// TIA Portal V20 export
// export: Created 2025-12-01T14:56:58.3126404Z, ExportSetting None, DisplayName Totally Integrated Automation Portal, DisplayVersion V20 Update 3, DisplayName TIA Portal Openness, DisplayVersion V20 Update 3, DisplayName TIA Portal Version Control Interface, DisplayVersion V20 Update 3, DisplayName STEP 7 Professional, DisplayVersion V20 Update 3, DisplayName STEP 7 Safety, DisplayVersion V20 Update 2, DisplayName WinCC Basic/Comfort/Advanced, DisplayVersion V20 Update 3, DisplayName WinCC Professional, DisplayVersion V20 Update 3, DisplayName WinCC Unified, DisplayVersion V20 Update 3
FUNCTION_BLOCK "FB87_GALIBO_3Frontales"   // FB87, LAD
TITLE = Galibo de 3 Desplomes Frontales (2024)
{ S7_Optimized_Access := 'FALSE' }
AUTHOR : GALIBO
NAME : 20140101
VERSION : 3.0
// stored: AutoNumber false, SetENOAutomatically false
   VAR_INPUT
      Mesa : UInt;
      NumGalibo : UInt;
      EnRodillos : Bool;
      pHs_LecturaDelantera_Des1 : Bool;
      pHs_LecturaTrasera_Des1 : Bool;
      pHs_LecturaDelantera_Des2 : Bool;
      pHs_LecturaTrasera_Des2 : Bool;
      pHs_LecturaDelantera_Error : Bool;
      pHs_LecturaTrasera_Error : Bool;
      pHs_Frontal_1 : Bool;
      pHs_Frontal_2 : Bool;
      pHs_Frontal_3 : Bool;
      HabilitarLectura : Bool;
      PermisoLectura : Bool;
      Rearmar_ConMesaLibre : Bool;
      Numero_Desplomes_2 : Bool;
      Numero_Desplomes_3 : Bool;
   END_VAR
   VAR_OUTPUT
      Baliza : Bool;
      ErrorFrontal : Bool;
      FinLectura : Bool;
   END_VAR
   VAR
      GAL_ET00 : Bool;
      GAL_ET01 : Bool;
      GAL_ET02 : Bool;
      GAL_ET03 : Bool;
      GAL_ET04 : Bool;
      pHsGalibo_OK { ExternalAccessible := 'False'; ExternalVisible := 'False'; ExternalWritable := 'False'} : Bool;
      pHsFrontal_OK : Bool;
      CaraDelantera_Des_PEQUEÑO_NOK : Bool;
      CaraTrasera_Des_PEQUEÑO_NOK : Bool;
      CaraDelantera_Des_MEDIANO_NOK : Bool;
      CaraTrasera_Des_MEDIANO_NOK : Bool;
      CaraDelantera_Des_NOK : Bool;
      CaraTrasera_Des_NOK : Bool;
      CodigoLargura : SInt;
      MemoCodigo : Word;
      STAT_Baliza_Galibo : Bool;
   END_VAR
   VAR_TEMP
      EstadoZona : "EstadoZona";
      EstadoVI : "EstadosMesa";
   END_VAR
   VAR_TEMP   // added for the SCL form of the ladder/FBD networks
      _w1 : Bool;
   END_VAR
BEGIN

REGION Network 1: INICIALIZAR - Recoger las Variables de Estado de la Mesa
   // Se recoge - Estado_CBx
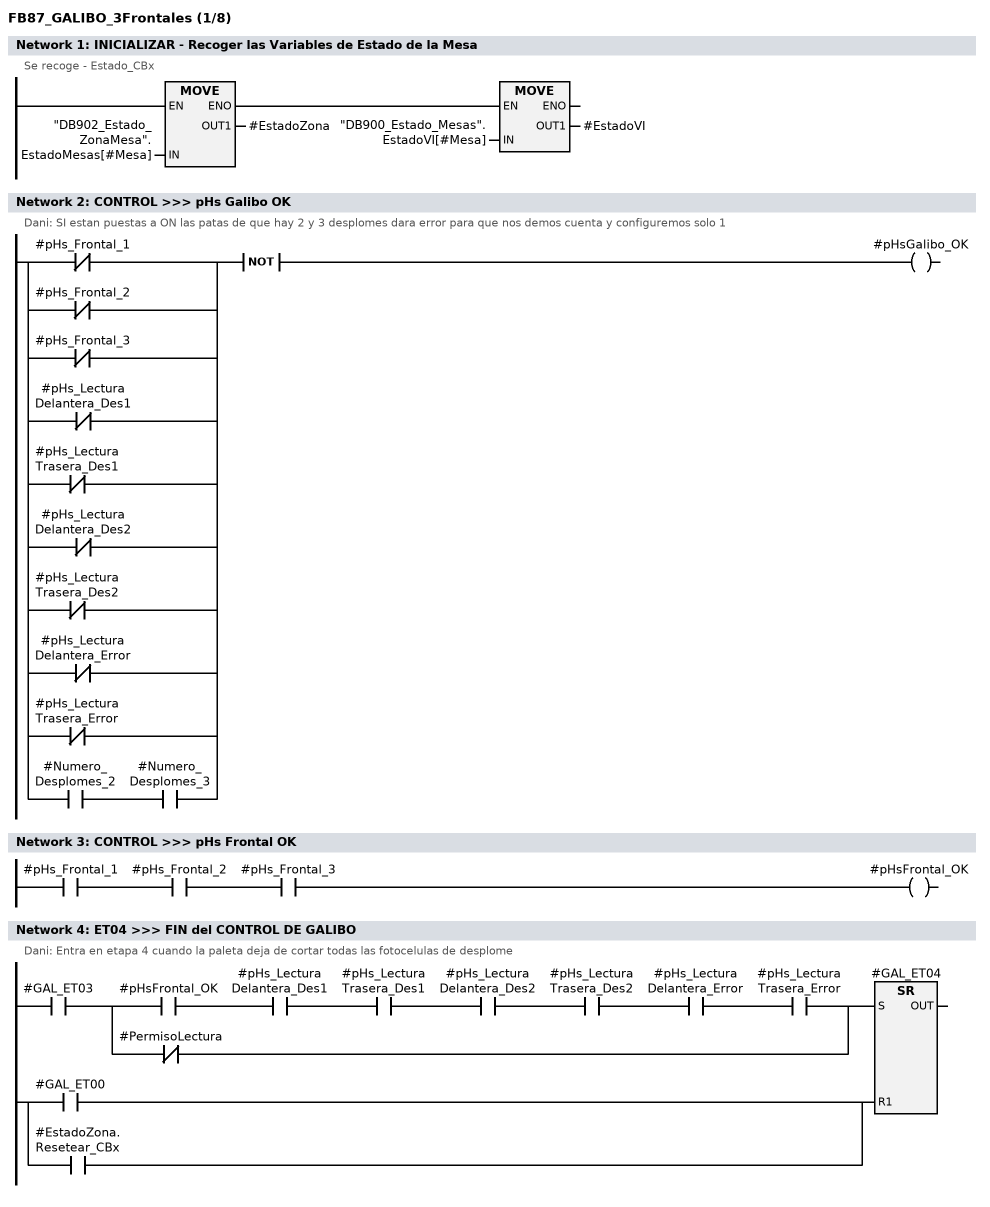
   RUNG wire#powerrail
      Move(in := "DB902_Estado_ZonaMesa".EstadoMesas[#Mesa], out1 => #EstadoZona)
      Move(in := "DB900_Estado_Mesas".EstadoVI[#Mesa], out1 => #EstadoVI)
   END_RUNG
   // the same network as SCL:
   #EstadoZona := "DB902_Estado_ZonaMesa".EstadoMesas[#Mesa];
   #EstadoVI := "DB900_Estado_Mesas".EstadoVI[#Mesa];
END_REGION

REGION Network 2: CONTROL >>> pHs Galibo OK
   // Dani: SI estan puestas a ON las patas de que hay 2 y 3 desplomes dara error para que nos demos cuenta y configuremos solo 1
   RUNG wire#powerrail
      I_Contact( #pHs_Frontal_1 )
      wire#w1
      Not()
      Coil( #pHsGalibo_OK )
   END_RUNG
   RUNG wire#powerrail
      I_Contact( #pHs_Frontal_2 )
   END_RUNG wire#w1
   RUNG wire#powerrail
      I_Contact( #pHs_Frontal_3 )
   END_RUNG wire#w1
   RUNG wire#powerrail
      I_Contact( #pHs_LecturaDelantera_Des1 )
   END_RUNG wire#w1
   RUNG wire#powerrail
      I_Contact( #pHs_LecturaTrasera_Des1 )
   END_RUNG wire#w1
   RUNG wire#powerrail
      I_Contact( #pHs_LecturaDelantera_Des2 )
   END_RUNG wire#w1
   RUNG wire#powerrail
      I_Contact( #pHs_LecturaTrasera_Des2 )
   END_RUNG wire#w1
   RUNG wire#powerrail
      I_Contact( #pHs_LecturaDelantera_Error )
   END_RUNG wire#w1
   RUNG wire#powerrail
      I_Contact( #pHs_LecturaTrasera_Error )
   END_RUNG wire#w1
   RUNG wire#powerrail
      Contact( #Numero_Desplomes_2 )
      Contact( #Numero_Desplomes_3 )
   END_RUNG wire#w1
   // the same network as SCL:
   #pHsGalibo_OK := NOT (NOT #pHs_Frontal_1 OR NOT #pHs_Frontal_2 OR NOT #pHs_Frontal_3 OR NOT #pHs_LecturaDelantera_Des1 OR NOT #pHs_LecturaTrasera_Des1 OR NOT #pHs_LecturaDelantera_Des2 OR NOT #pHs_LecturaTrasera_Des2 OR NOT #pHs_LecturaDelantera_Error OR NOT #pHs_LecturaTrasera_Error OR (#Numero_Desplomes_2 AND #Numero_Desplomes_3));
END_REGION

REGION Network 3: CONTROL >>> pHs Frontal OK
   RUNG wire#powerrail
      Contact( #pHs_Frontal_1 )
      Contact( #pHs_Frontal_2 )
      Contact( #pHs_Frontal_3 )
      Coil( #pHsFrontal_OK )
   END_RUNG
   // the same network as SCL:
   #pHsFrontal_OK := #pHs_Frontal_1 AND #pHs_Frontal_2 AND #pHs_Frontal_3;
END_REGION

REGION Network 4: ET04 >>> FIN del CONTROL DE GALIBO
   // Dani: Entra en etapa 4 cuando la paleta deja de cortar todas las fotocelulas de desplome
   RUNG wire#powerrail
      Contact( #GAL_ET03 )
      wire#w1
      Contact( #pHsFrontal_OK )
      Contact( #pHs_LecturaDelantera_Des1 )
      Contact( #pHs_LecturaTrasera_Des1 )
      Contact( #pHs_LecturaDelantera_Des2 )
      Contact( #pHs_LecturaTrasera_Des2 )
      Contact( #pHs_LecturaDelantera_Error )
      Contact( #pHs_LecturaTrasera_Error )
      wire#w2
      S_SR(operand := #GAL_ET04, r1 := wire#w3)
   END_RUNG
   RUNG wire#w1
      I_Contact( #PermisoLectura )
   END_RUNG wire#w2
   RUNG wire#powerrail
      Contact( #GAL_ET00 )
   END_RUNG wire#w3
   RUNG wire#powerrail
      Contact( #EstadoZona.Resetear_CBx )
   END_RUNG wire#w3
   // the same network as SCL:
   IF #GAL_ET03 AND ((#pHsFrontal_OK AND #pHs_LecturaDelantera_Des1 AND #pHs_LecturaTrasera_Des1 AND #pHs_LecturaDelantera_Des2 AND #pHs_LecturaTrasera_Des2 AND #pHs_LecturaDelantera_Error AND #pHs_LecturaTrasera_Error) OR NOT #PermisoLectura) THEN
       #GAL_ET04 := TRUE;   // SR flip-flop
   END_IF;
   IF #GAL_ET00 OR #EstadoZona.Resetear_CBx THEN #GAL_ET04 := FALSE; END_IF;
END_REGION

REGION Network 5: ET03 >>> Lectura de CARA TRASERA
   // Dani: Entra en etapa 3 cuando la paleta corta una de las fotocelula de desplomeque esten configuradas
   // En la fotocelula error siempre estara metido el desplome mayor tengamos 1, 2 o 3 desplomes
   // En la fotocelula desplome 2 solo tendremos metido el desplome mediano si el numero de desplome es 3
   // En la fotocelula desplome 1 tendremos metido el desplome mas pequeño si el numero de desplome es 2 o 3.
   // Como los desplomes que no existan estaran siempre a ON no hace falta programar ningun tipo de logica para saber cuando se corta la primera
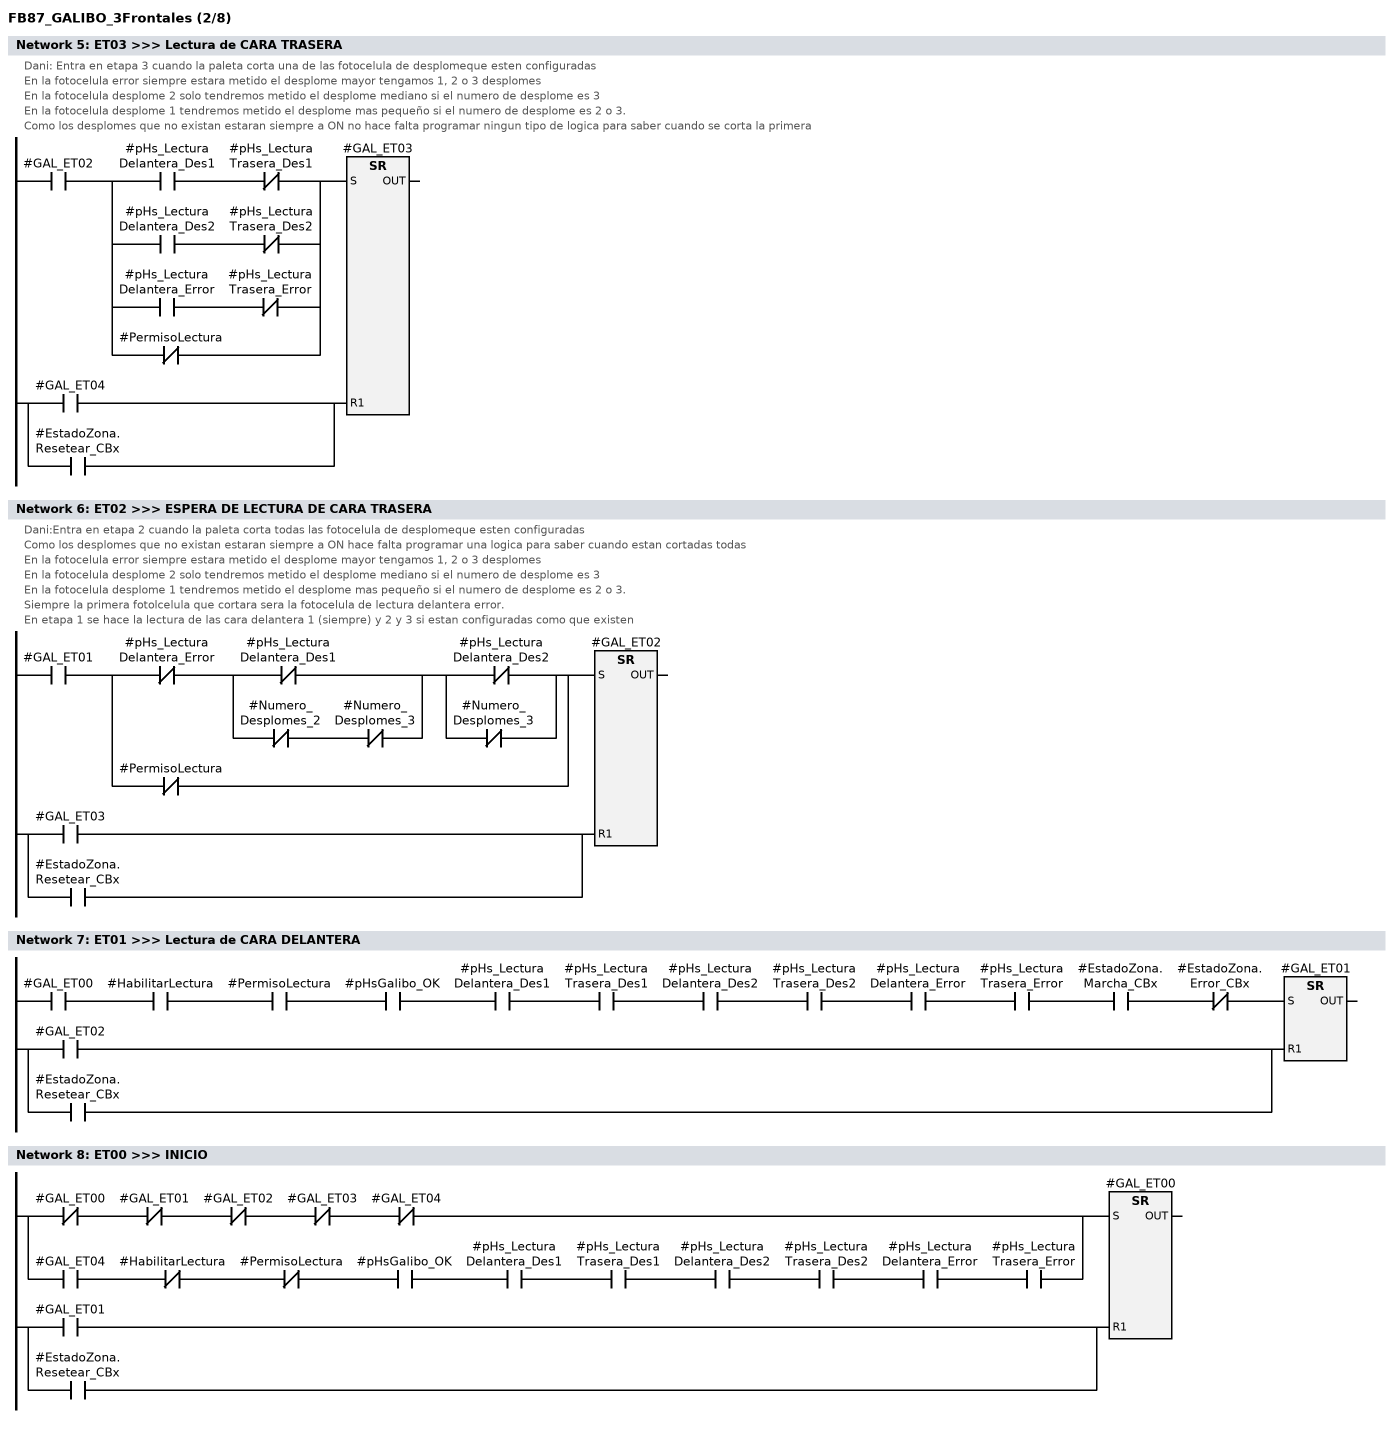
   RUNG wire#powerrail
      Contact( #GAL_ET02 )
      wire#w1
      Contact( #pHs_LecturaDelantera_Des1 )
      I_Contact( #pHs_LecturaTrasera_Des1 )
      wire#w2
      S_SR(operand := #GAL_ET03, r1 := wire#w3)
   END_RUNG
   RUNG wire#w1
      Contact( #pHs_LecturaDelantera_Des2 )
      I_Contact( #pHs_LecturaTrasera_Des2 )
   END_RUNG wire#w2
   RUNG wire#w1
      Contact( #pHs_LecturaDelantera_Error )
      I_Contact( #pHs_LecturaTrasera_Error )
   END_RUNG wire#w2
   RUNG wire#w1
      I_Contact( #PermisoLectura )
   END_RUNG wire#w2
   RUNG wire#powerrail
      Contact( #GAL_ET04 )
   END_RUNG wire#w3
   RUNG wire#powerrail
      Contact( #EstadoZona.Resetear_CBx )
   END_RUNG wire#w3
   // the same network as SCL:
   IF #GAL_ET02 AND ((#pHs_LecturaDelantera_Des1 AND NOT #pHs_LecturaTrasera_Des1) OR (#pHs_LecturaDelantera_Des2 AND NOT #pHs_LecturaTrasera_Des2) OR (#pHs_LecturaDelantera_Error AND NOT #pHs_LecturaTrasera_Error) OR NOT #PermisoLectura) THEN
       #GAL_ET03 := TRUE;   // SR flip-flop
   END_IF;
   IF #GAL_ET04 OR #EstadoZona.Resetear_CBx THEN #GAL_ET03 := FALSE; END_IF;
END_REGION

REGION Network 6: ET02 >>> ESPERA DE LECTURA DE CARA TRASERA
   // Dani:Entra en etapa 2 cuando la paleta corta todas las fotocelula de desplomeque esten configuradas
   // Como los desplomes que no existan estaran siempre a ON hace falta programar una logica para saber cuando estan cortadas todas
   // En la fotocelula error siempre estara metido el desplome mayor tengamos 1, 2 o 3 desplomes
   // En la fotocelula desplome 2 solo tendremos metido el desplome mediano si el numero de desplome es 3
   // En la fotocelula desplome 1 tendremos metido el desplome mas pequeño si el numero de desplome es 2 o 3.
   // Siempre la primera fotolcelula que cortara sera la fotocelula de lectura delantera error.
   // En etapa 1 se hace la lectura de las cara delantera 1 (siempre) y 2 y 3 si estan configuradas como que existen
   RUNG wire#powerrail
      Contact( #GAL_ET01 )
      wire#w1
      I_Contact( #pHs_LecturaDelantera_Error )
      wire#w2
      I_Contact( #pHs_LecturaDelantera_Des1 )
      wire#w3
      I_Contact( #pHs_LecturaDelantera_Des2 )
      wire#w4
      S_SR(operand := #GAL_ET02, r1 := wire#w5)
   END_RUNG
   RUNG wire#w2
      I_Contact( #Numero_Desplomes_2 )
      I_Contact( #Numero_Desplomes_3 )
   END_RUNG wire#w3
   RUNG wire#w3
      I_Contact( #Numero_Desplomes_3 )
   END_RUNG wire#w4
   RUNG wire#w1
      I_Contact( #PermisoLectura )
   END_RUNG wire#w4
   RUNG wire#powerrail
      Contact( #GAL_ET03 )
   END_RUNG wire#w5
   RUNG wire#powerrail
      Contact( #EstadoZona.Resetear_CBx )
   END_RUNG wire#w5
   // the same network as SCL:
   IF #GAL_ET01 AND ((NOT #pHs_LecturaDelantera_Error AND (NOT #pHs_LecturaDelantera_Des1 OR (NOT #Numero_Desplomes_2 AND NOT #Numero_Desplomes_3)) AND (NOT #pHs_LecturaDelantera_Des2 OR NOT #Numero_Desplomes_3)) OR NOT #PermisoLectura) THEN
       #GAL_ET02 := TRUE;   // SR flip-flop
   END_IF;
   IF #GAL_ET03 OR #EstadoZona.Resetear_CBx THEN #GAL_ET02 := FALSE; END_IF;
END_REGION

REGION Network 7: ET01 >>> Lectura de CARA DELANTERA
   RUNG wire#powerrail
      Contact( #GAL_ET00 )
      Contact( #HabilitarLectura )
      Contact( #PermisoLectura )
      Contact( #pHsGalibo_OK )
      Contact( #pHs_LecturaDelantera_Des1 )
      Contact( #pHs_LecturaTrasera_Des1 )
      Contact( #pHs_LecturaDelantera_Des2 )
      Contact( #pHs_LecturaTrasera_Des2 )
      Contact( #pHs_LecturaDelantera_Error )
      Contact( #pHs_LecturaTrasera_Error )
      Contact( #EstadoZona.Marcha_CBx )
      I_Contact( #EstadoZona.Error_CBx )
      S_SR(operand := #GAL_ET01, r1 := wire#w1)
   END_RUNG
   RUNG wire#powerrail
      Contact( #GAL_ET02 )
   END_RUNG wire#w1
   RUNG wire#powerrail
      Contact( #EstadoZona.Resetear_CBx )
   END_RUNG wire#w1
   // the same network as SCL:
   IF #GAL_ET00 AND #HabilitarLectura AND #PermisoLectura AND #pHsGalibo_OK AND #pHs_LecturaDelantera_Des1 AND #pHs_LecturaTrasera_Des1 AND #pHs_LecturaDelantera_Des2 AND #pHs_LecturaTrasera_Des2 AND #pHs_LecturaDelantera_Error AND #pHs_LecturaTrasera_Error AND #EstadoZona.Marcha_CBx AND NOT #EstadoZona.Error_CBx THEN
       #GAL_ET01 := TRUE;   // SR flip-flop
   END_IF;
   IF #GAL_ET02 OR #EstadoZona.Resetear_CBx THEN #GAL_ET01 := FALSE; END_IF;
END_REGION

REGION Network 8: ET00 >>> INICIO
   RUNG wire#powerrail
      I_Contact( #GAL_ET00 )
      I_Contact( #GAL_ET01 )
      I_Contact( #GAL_ET02 )
      I_Contact( #GAL_ET03 )
      I_Contact( #GAL_ET04 )
      wire#w1
      S_SR(operand := #GAL_ET00, r1 := wire#w2)
   END_RUNG
   RUNG wire#powerrail
      Contact( #GAL_ET04 )
      I_Contact( #HabilitarLectura )
      I_Contact( #PermisoLectura )
      Contact( #pHsGalibo_OK )
      Contact( #pHs_LecturaDelantera_Des1 )
      Contact( #pHs_LecturaTrasera_Des1 )
      Contact( #pHs_LecturaDelantera_Des2 )
      Contact( #pHs_LecturaTrasera_Des2 )
      Contact( #pHs_LecturaDelantera_Error )
      Contact( #pHs_LecturaTrasera_Error )
   END_RUNG wire#w1
   RUNG wire#powerrail
      Contact( #GAL_ET01 )
   END_RUNG wire#w2
   RUNG wire#powerrail
      Contact( #EstadoZona.Resetear_CBx )
   END_RUNG wire#w2
   // the same network as SCL:
   IF (NOT #GAL_ET00 AND NOT #GAL_ET01 AND NOT #GAL_ET02 AND NOT #GAL_ET03 AND NOT #GAL_ET04) OR (#GAL_ET04 AND NOT #HabilitarLectura AND NOT #PermisoLectura AND #pHsGalibo_OK AND #pHs_LecturaDelantera_Des1 AND #pHs_LecturaTrasera_Des1 AND #pHs_LecturaDelantera_Des2 AND #pHs_LecturaTrasera_Des2 AND #pHs_LecturaDelantera_Error AND #pHs_LecturaTrasera_Error) THEN
       #GAL_ET00 := TRUE;   // SR flip-flop
   END_IF;
   IF #GAL_ET01 OR #EstadoZona.Resetear_CBx THEN #GAL_ET00 := FALSE; END_IF;
END_REGION

REGION Network 9: ERROR >>> Fotocelulas de Galibo
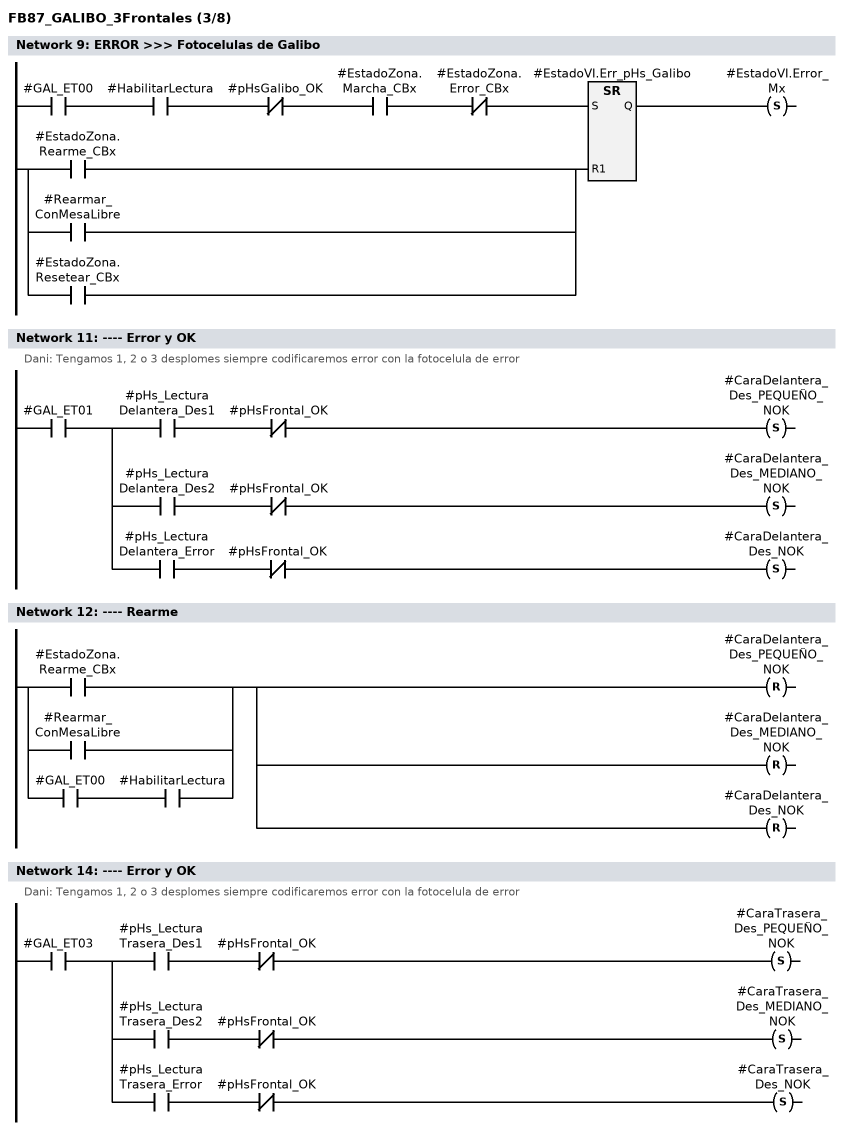
   RUNG wire#powerrail
      Contact( #GAL_ET00 )
      Contact( #HabilitarLectura )
      I_Contact( #pHsGalibo_OK )
      Contact( #EstadoZona.Marcha_CBx )
      I_Contact( #EstadoZona.Error_CBx )
      S_SR(operand := #EstadoVI.Err_pHs_Galibo, r1 := wire#w1)
      S_Coil( #EstadoVI.Error_Mx )
   END_RUNG
   RUNG wire#powerrail
      Contact( #EstadoZona.Rearme_CBx )
   END_RUNG wire#w1
   RUNG wire#powerrail
      Contact( #Rearmar_ConMesaLibre )
   END_RUNG wire#w1
   RUNG wire#powerrail
      Contact( #EstadoZona.Resetear_CBx )
   END_RUNG wire#w1
   // the same network as SCL:
   IF #GAL_ET00 AND #HabilitarLectura AND NOT #pHsGalibo_OK AND #EstadoZona.Marcha_CBx AND NOT #EstadoZona.Error_CBx THEN
       #EstadoVI.Err_pHs_Galibo := TRUE;   // SR flip-flop
   END_IF;
   IF #EstadoZona.Rearme_CBx OR #Rearmar_ConMesaLibre OR #EstadoZona.Resetear_CBx THEN
       #EstadoVI.Err_pHs_Galibo := FALSE;
   END_IF;
   IF #EstadoVI.Err_pHs_Galibo THEN #EstadoVI.Error_Mx := TRUE; END_IF;
END_REGION

REGION Network 10: VARIABLES DE CONTROL DE LARGURA >>> Activar la lectura de Cara Delantera
END_REGION

REGION Network 11: ---- Error y OK
   // Dani: Tengamos 1, 2 o 3 desplomes siempre codificaremos error con la fotocelula de error
   RUNG wire#powerrail
      Contact( #GAL_ET01 )
      wire#w1
      Contact( #pHs_LecturaDelantera_Des1 )
      I_Contact( #pHsFrontal_OK )
      S_Coil( #CaraDelantera_Des_PEQUEÑO_NOK )
   END_RUNG
   RUNG wire#w1
      Contact( #pHs_LecturaDelantera_Des2 )
      I_Contact( #pHsFrontal_OK )
      S_Coil( #CaraDelantera_Des_MEDIANO_NOK )
   END_RUNG
   RUNG wire#w1
      Contact( #pHs_LecturaDelantera_Error )
      I_Contact( #pHsFrontal_OK )
      S_Coil( #CaraDelantera_Des_NOK )
   END_RUNG
   // the same network as SCL:
   IF #GAL_ET01 AND #pHs_LecturaDelantera_Des1 AND NOT #pHsFrontal_OK THEN
       #CaraDelantera_Des_PEQUEÑO_NOK := TRUE;
   END_IF;
   IF #GAL_ET01 AND #pHs_LecturaDelantera_Des2 AND NOT #pHsFrontal_OK THEN
       #CaraDelantera_Des_MEDIANO_NOK := TRUE;
   END_IF;
   IF #GAL_ET01 AND #pHs_LecturaDelantera_Error AND NOT #pHsFrontal_OK THEN
       #CaraDelantera_Des_NOK := TRUE;
   END_IF;
END_REGION

REGION Network 12: ---- Rearme
   RUNG wire#powerrail
      Contact( #EstadoZona.Rearme_CBx )
      wire#w1
      R_Coil( #CaraDelantera_Des_PEQUEÑO_NOK )
   END_RUNG
   RUNG wire#powerrail
      Contact( #Rearmar_ConMesaLibre )
   END_RUNG wire#w1
   RUNG wire#powerrail
      Contact( #GAL_ET00 )
      Contact( #HabilitarLectura )
   END_RUNG wire#w1
   RUNG wire#w1
      R_Coil( #CaraDelantera_Des_MEDIANO_NOK )
   END_RUNG
   RUNG wire#w1
      R_Coil( #CaraDelantera_Des_NOK )
   END_RUNG
   // the same network as SCL:
   IF #EstadoZona.Rearme_CBx OR #Rearmar_ConMesaLibre OR (#GAL_ET00 AND #HabilitarLectura) THEN
       #CaraDelantera_Des_PEQUEÑO_NOK := FALSE;
       #CaraDelantera_Des_MEDIANO_NOK := FALSE;
       #CaraDelantera_Des_NOK := FALSE;
   END_IF;
END_REGION

REGION Network 13: VARIABLES DE CONTROL DE LARGURA >>> Activar la lectura de Cara Trasera
END_REGION

REGION Network 14: ---- Error y OK
   // Dani: Tengamos 1, 2 o 3 desplomes siempre codificaremos error con la fotocelula de error
   RUNG wire#powerrail
      Contact( #GAL_ET03 )
      wire#w1
      Contact( #pHs_LecturaTrasera_Des1 )
      I_Contact( #pHsFrontal_OK )
      S_Coil( #CaraTrasera_Des_PEQUEÑO_NOK )
   END_RUNG
   RUNG wire#w1
      Contact( #pHs_LecturaTrasera_Des2 )
      I_Contact( #pHsFrontal_OK )
      S_Coil( #CaraTrasera_Des_MEDIANO_NOK )
   END_RUNG
   RUNG wire#w1
      Contact( #pHs_LecturaTrasera_Error )
      I_Contact( #pHsFrontal_OK )
      S_Coil( #CaraTrasera_Des_NOK )
   END_RUNG
   // the same network as SCL:
   IF #GAL_ET03 AND #pHs_LecturaTrasera_Des1 AND NOT #pHsFrontal_OK THEN
       #CaraTrasera_Des_PEQUEÑO_NOK := TRUE;
   END_IF;
   IF #GAL_ET03 AND #pHs_LecturaTrasera_Des2 AND NOT #pHsFrontal_OK THEN
       #CaraTrasera_Des_MEDIANO_NOK := TRUE;
   END_IF;
   IF #GAL_ET03 AND #pHs_LecturaTrasera_Error AND NOT #pHsFrontal_OK THEN
       #CaraTrasera_Des_NOK := TRUE;
   END_IF;
END_REGION

REGION Network 15: ---- Rearme
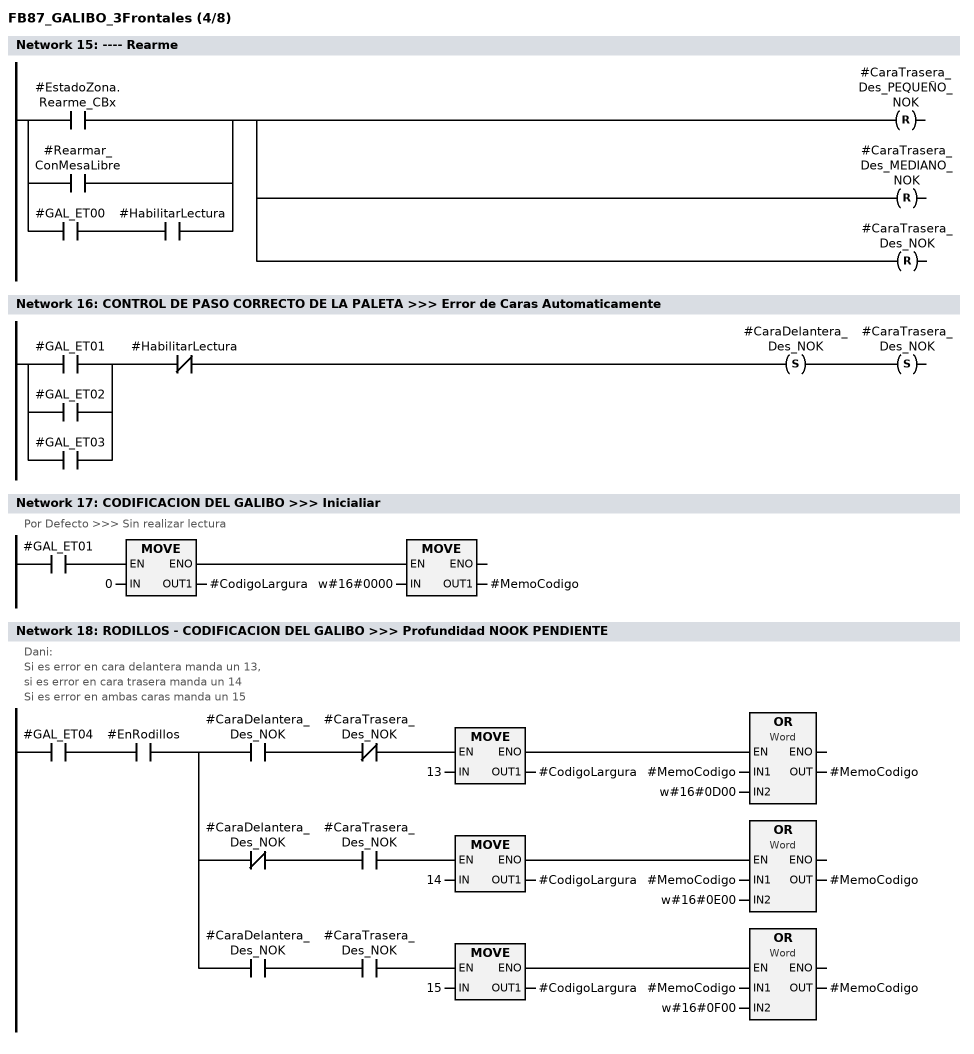
   RUNG wire#powerrail
      Contact( #EstadoZona.Rearme_CBx )
      wire#w1
      R_Coil( #CaraTrasera_Des_PEQUEÑO_NOK )
   END_RUNG
   RUNG wire#powerrail
      Contact( #Rearmar_ConMesaLibre )
   END_RUNG wire#w1
   RUNG wire#powerrail
      Contact( #GAL_ET00 )
      Contact( #HabilitarLectura )
   END_RUNG wire#w1
   RUNG wire#w1
      R_Coil( #CaraTrasera_Des_MEDIANO_NOK )
   END_RUNG
   RUNG wire#w1
      R_Coil( #CaraTrasera_Des_NOK )
   END_RUNG
   // the same network as SCL:
   IF #EstadoZona.Rearme_CBx OR #Rearmar_ConMesaLibre OR (#GAL_ET00 AND #HabilitarLectura) THEN
       #CaraTrasera_Des_PEQUEÑO_NOK := FALSE;
       #CaraTrasera_Des_MEDIANO_NOK := FALSE;
       #CaraTrasera_Des_NOK := FALSE;
   END_IF;
END_REGION

REGION Network 16: CONTROL DE PASO CORRECTO DE LA PALETA >>> Error de Caras Automaticamente
   RUNG wire#powerrail
      Contact( #GAL_ET01 )
      wire#w1
      I_Contact( #HabilitarLectura )
      S_Coil( #CaraDelantera_Des_NOK )
      S_Coil( #CaraTrasera_Des_NOK )
   END_RUNG
   RUNG wire#powerrail
      Contact( #GAL_ET02 )
   END_RUNG wire#w1
   RUNG wire#powerrail
      Contact( #GAL_ET03 )
   END_RUNG wire#w1
   // the same network as SCL:
   IF (#GAL_ET01 OR #GAL_ET02 OR #GAL_ET03) AND NOT #HabilitarLectura THEN
       #CaraDelantera_Des_NOK := TRUE;
       #CaraTrasera_Des_NOK := TRUE;
   END_IF;
END_REGION

REGION Network 17: CODIFICACION DEL GALIBO >>> Inicialiar
   // Por Defecto >>> Sin realizar lectura
   RUNG wire#powerrail
      Contact( #GAL_ET01 )
      { S7_GenerateENO := "TRUE" } Move(in := 0, out1 => #CodigoLargura)
      { S7_GenerateENO := "TRUE" } Move(in := w#16#0000, out1 => #MemoCodigo)
   END_RUNG
   // the same network as SCL:
   // ENO of a box is taken as its EN; it also drops when the box reports an error
   IF #GAL_ET01 THEN
       #CodigoLargura := 0;
       #MemoCodigo := w#16#0000;
   END_IF;
END_REGION

REGION Network 18: RODILLOS - CODIFICACION DEL GALIBO >>> Profundidad NOOK PENDIENTE
   // Dani:
   // Si es error en cara delantera manda un 13, 
   // si es error en cara trasera manda un 14
   // Si es error en ambas caras manda un 15
   #_w1 := #GAL_ET04 AND #EnRodillos;
   IF #_w1 AND #CaraDelantera_Des_NOK AND NOT #CaraTrasera_Des_NOK THEN
       #CodigoLargura := 13;
       #MemoCodigo := #MemoCodigo OR w#16#0D00;
   END_IF;
   IF #_w1 AND NOT #CaraDelantera_Des_NOK AND #CaraTrasera_Des_NOK THEN
       #CodigoLargura := 14;
       #MemoCodigo := #MemoCodigo OR w#16#0E00;
   END_IF;
   IF #_w1 AND #CaraDelantera_Des_NOK AND #CaraTrasera_Des_NOK THEN
       #CodigoLargura := 15;
       #MemoCodigo := #MemoCodigo OR w#16#0F00;
   END_IF;
END_REGION

REGION Network 19: RODILLOS - CODIFICACION DEL GALIBO >>> Profundidad OK - Codificacion
   // Dani:  los Nook solo se escriben si el desplome esta configurado
   // si hay 1 desplome envia 1 si la carga no da error de desplome
   // Si hay 2 desplomes envia 1 si no hay desplome pequeño y 2 si no hay error de desplome
   // Si hay 3 desplomes envia 1 si no hay desplome pequeño, 2 si no hay desplome mediano y 3 si no hay error de desplome
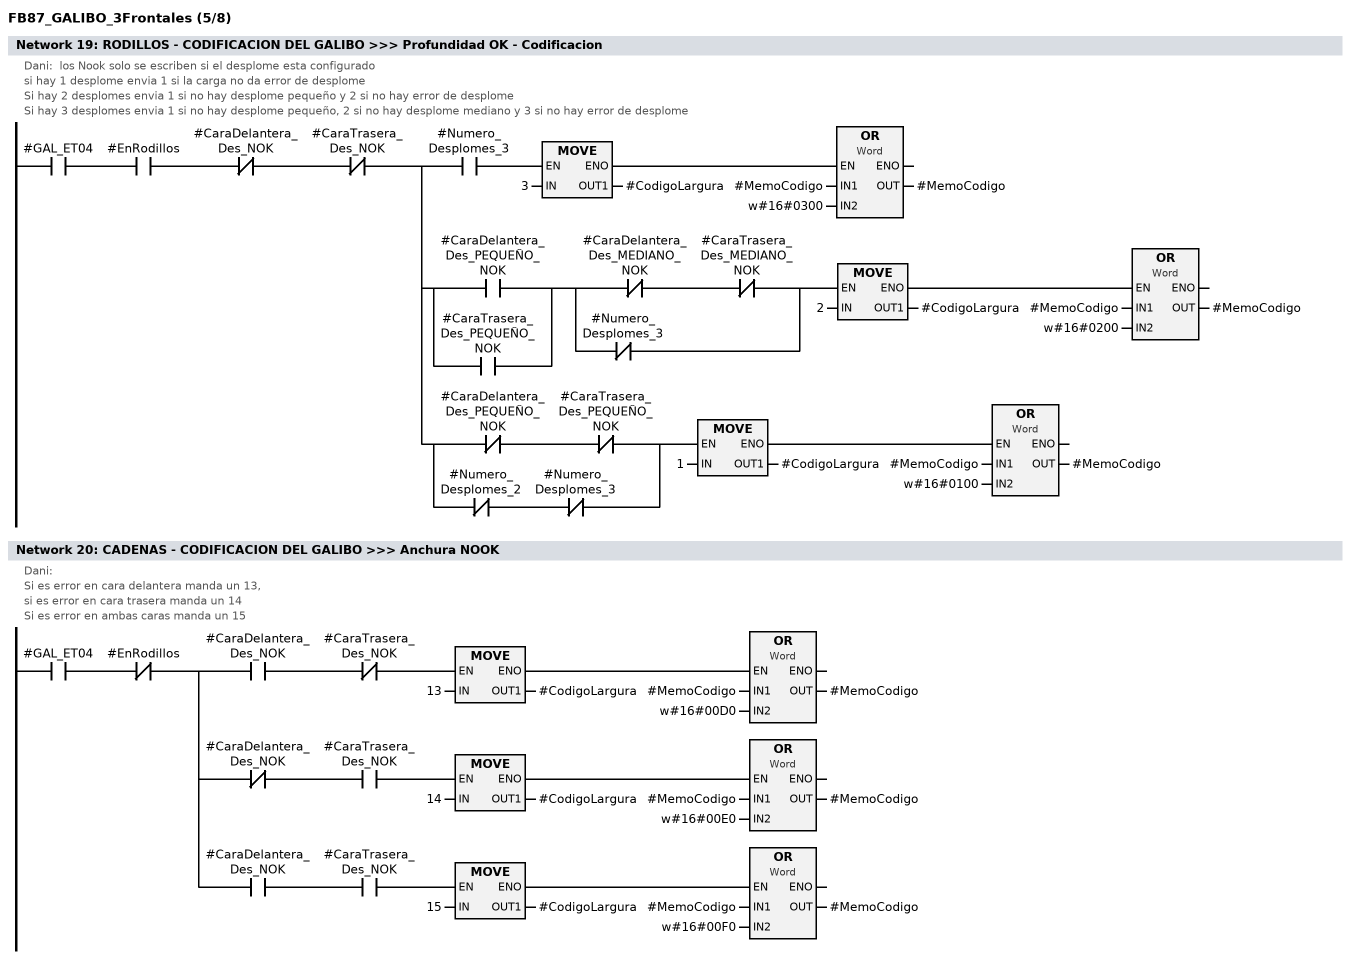
   #_w1 := #GAL_ET04 AND #EnRodillos AND NOT #CaraDelantera_Des_NOK AND NOT #CaraTrasera_Des_NOK;
   IF #_w1 AND #Numero_Desplomes_3 THEN
       #CodigoLargura := 3;
       #MemoCodigo := #MemoCodigo OR w#16#0300;
   END_IF;
   IF #_w1 AND (#CaraDelantera_Des_PEQUEÑO_NOK OR #CaraTrasera_Des_PEQUEÑO_NOK) AND ((NOT #CaraDelantera_Des_MEDIANO_NOK AND NOT #CaraTrasera_Des_MEDIANO_NOK) OR NOT #Numero_Desplomes_3) THEN
       #CodigoLargura := 2;
       #MemoCodigo := #MemoCodigo OR w#16#0200;
   END_IF;
   IF #_w1 AND ((NOT #CaraDelantera_Des_PEQUEÑO_NOK AND NOT #CaraTrasera_Des_PEQUEÑO_NOK) OR (NOT #Numero_Desplomes_2 AND NOT #Numero_Desplomes_3)) THEN
       #CodigoLargura := 1;
       #MemoCodigo := #MemoCodigo OR w#16#0100;
   END_IF;
END_REGION

REGION Network 20: CADENAS - CODIFICACION DEL GALIBO >>> Anchura NOOK
   // Dani:
   // Si es error en cara delantera manda un 13, 
   // si es error en cara trasera manda un 14
   // Si es error en ambas caras manda un 15
   #_w1 := #GAL_ET04 AND NOT #EnRodillos;
   IF #_w1 AND #CaraDelantera_Des_NOK AND NOT #CaraTrasera_Des_NOK THEN
       #CodigoLargura := 13;
       #MemoCodigo := #MemoCodigo OR w#16#00D0;
   END_IF;
   IF #_w1 AND NOT #CaraDelantera_Des_NOK AND #CaraTrasera_Des_NOK THEN
       #CodigoLargura := 14;
       #MemoCodigo := #MemoCodigo OR w#16#00E0;
   END_IF;
   IF #_w1 AND #CaraDelantera_Des_NOK AND #CaraTrasera_Des_NOK THEN
       #CodigoLargura := 15;
       #MemoCodigo := #MemoCodigo OR w#16#00F0;
   END_IF;
END_REGION

REGION Network 21: CADENAS - CODIFICACION DEL GALIBO >>> Anchura OK - Codificacion
   // Dani:
   // Si la cargaes menor que desplome 1 manda 1
   // si la carga es mayor que desplome 1 y menor que desplome 2 manda 2
   // si la carga es mayor que desplome 2 y menor que desplome 3 manda 3
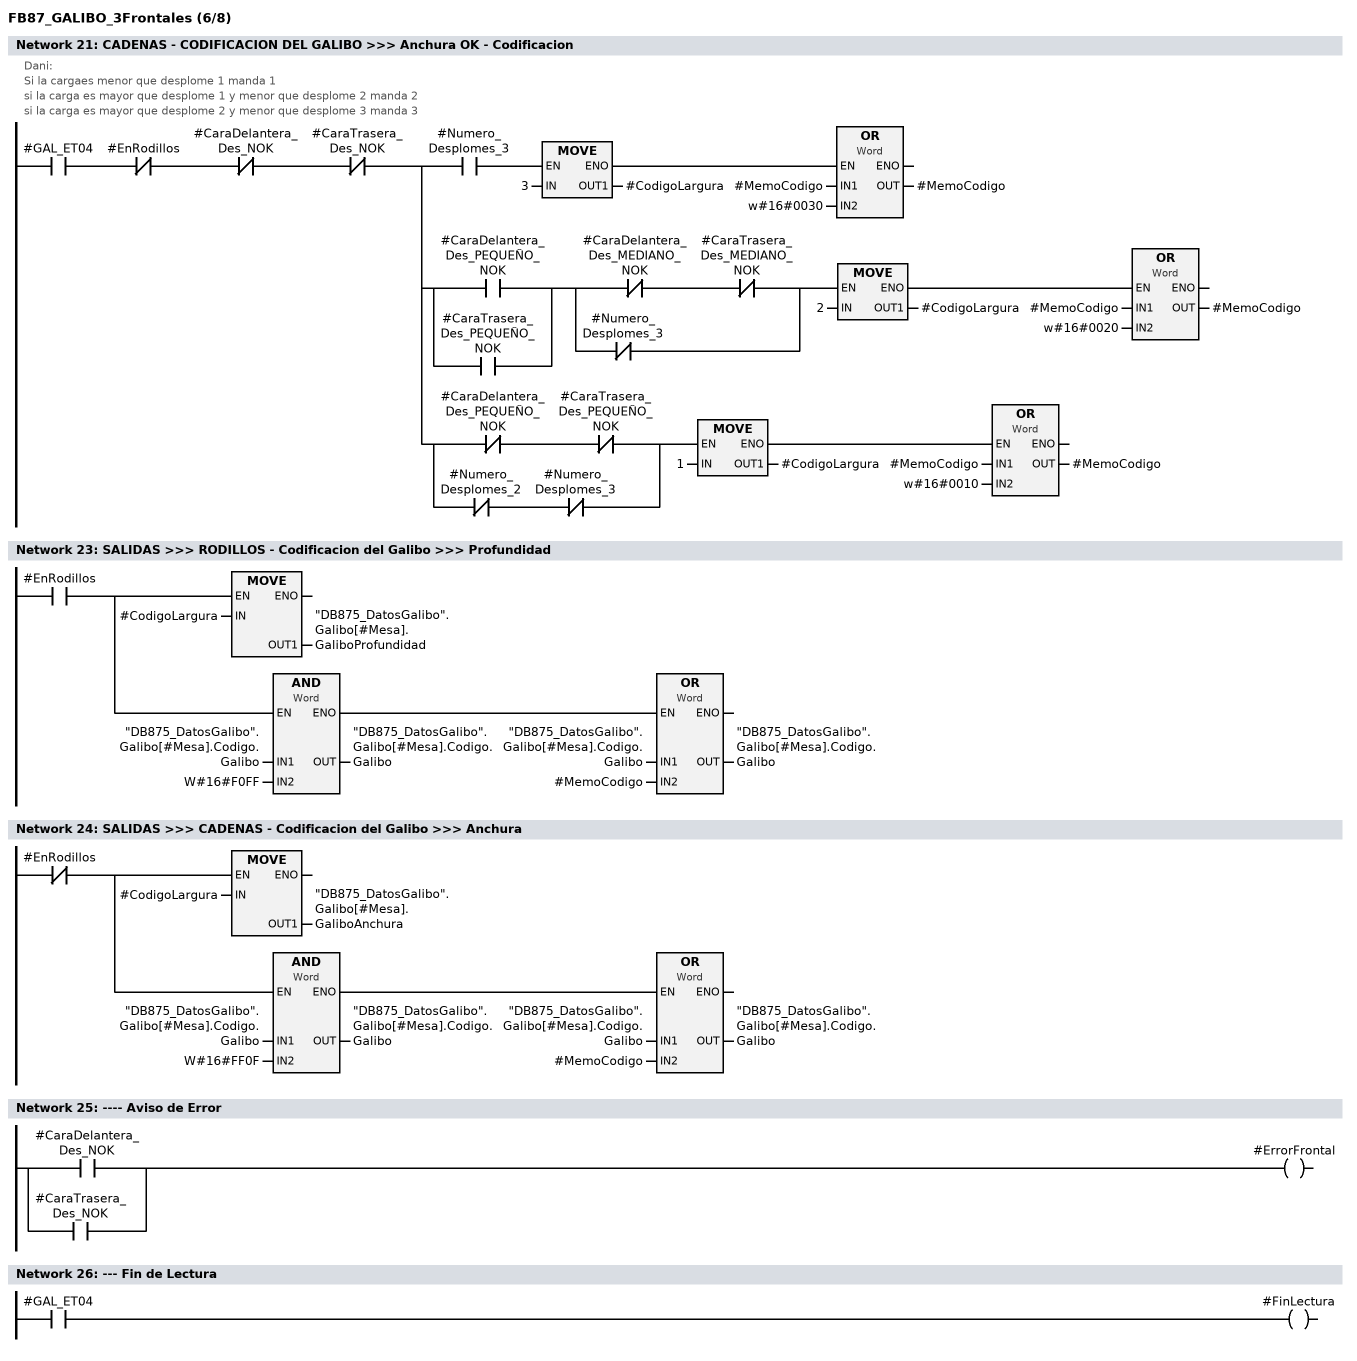
   #_w1 := #GAL_ET04 AND NOT #EnRodillos AND NOT #CaraDelantera_Des_NOK AND NOT #CaraTrasera_Des_NOK;
   IF #_w1 AND #Numero_Desplomes_3 THEN
       #CodigoLargura := 3;
       #MemoCodigo := #MemoCodigo OR w#16#0030;
   END_IF;
   IF #_w1 AND (#CaraDelantera_Des_PEQUEÑO_NOK OR #CaraTrasera_Des_PEQUEÑO_NOK) AND ((NOT #CaraDelantera_Des_MEDIANO_NOK AND NOT #CaraTrasera_Des_MEDIANO_NOK) OR NOT #Numero_Desplomes_3) THEN
       #CodigoLargura := 2;
       #MemoCodigo := #MemoCodigo OR w#16#0020;
   END_IF;
   IF #_w1 AND ((NOT #CaraDelantera_Des_PEQUEÑO_NOK AND NOT #CaraTrasera_Des_PEQUEÑO_NOK) OR (NOT #Numero_Desplomes_2 AND NOT #Numero_Desplomes_3)) THEN
       #CodigoLargura := 1;
       #MemoCodigo := #MemoCodigo OR w#16#0010;
   END_IF;
END_REGION

REGION Network 22: SALIDAS >>> Codificacion del Galibo y Error de Anchura
END_REGION

REGION Network 23: SALIDAS >>> RODILLOS - Codificacion del Galibo >>> Profundidad
   IF #EnRodillos THEN
       "DB875_DatosGalibo".Galibo[#Mesa].GaliboProfundidad := #CodigoLargura;
       "DB875_DatosGalibo".Galibo[#Mesa].Codigo.Galibo := "DB875_DatosGalibo".Galibo[#Mesa].Codigo.Galibo AND W#16#F0FF;
       "DB875_DatosGalibo".Galibo[#Mesa].Codigo.Galibo := "DB875_DatosGalibo".Galibo[#Mesa].Codigo.Galibo OR #MemoCodigo;
   END_IF;
END_REGION

REGION Network 24: SALIDAS >>> CADENAS - Codificacion del Galibo >>> Anchura
   IF NOT #EnRodillos THEN
       "DB875_DatosGalibo".Galibo[#Mesa].GaliboAnchura := #CodigoLargura;
       "DB875_DatosGalibo".Galibo[#Mesa].Codigo.Galibo := "DB875_DatosGalibo".Galibo[#Mesa].Codigo.Galibo AND W#16#FF0F;
       "DB875_DatosGalibo".Galibo[#Mesa].Codigo.Galibo := "DB875_DatosGalibo".Galibo[#Mesa].Codigo.Galibo OR #MemoCodigo;
   END_IF;
END_REGION

REGION Network 25: ---- Aviso de Error
   RUNG wire#powerrail
      Contact( #CaraDelantera_Des_NOK )
      wire#w1
      Coil( #ErrorFrontal )
   END_RUNG
   RUNG wire#powerrail
      Contact( #CaraTrasera_Des_NOK )
   END_RUNG wire#w1
   // the same network as SCL:
   #ErrorFrontal := #CaraDelantera_Des_NOK OR #CaraTrasera_Des_NOK;
END_REGION

REGION Network 26: --- Fin de Lectura
   RUNG wire#powerrail
      Contact( #GAL_ET04 )
      Coil( #FinLectura )
   END_RUNG
   // the same network as SCL:
   #FinLectura := #GAL_ET04;
END_REGION

REGION Network 27: SALIDAS >>> BALIZA
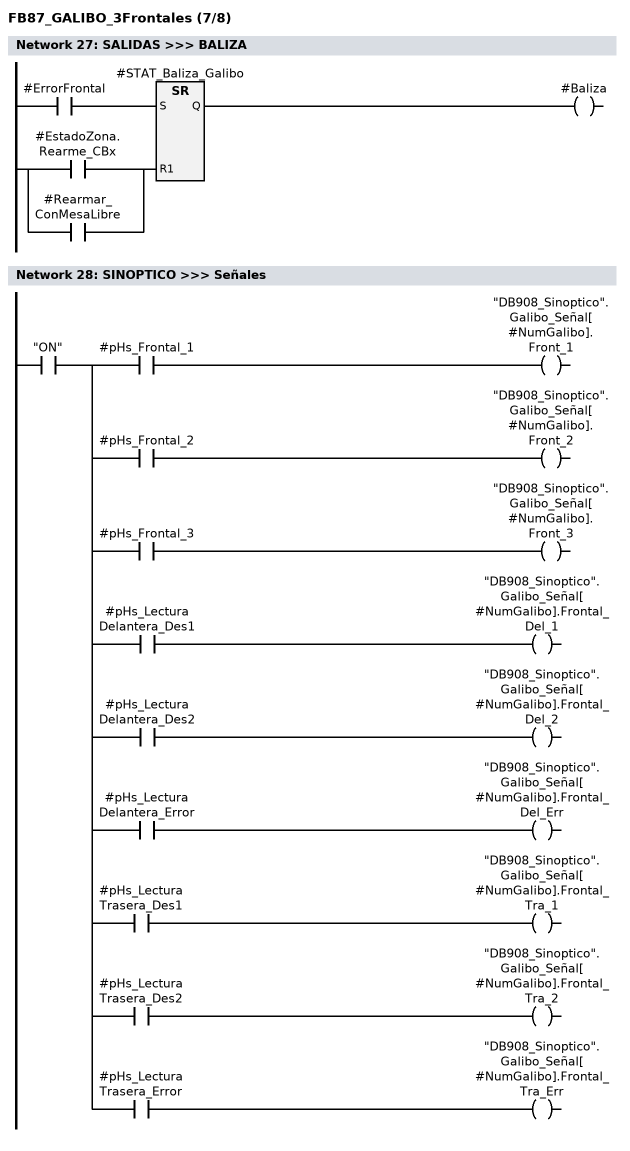
   RUNG wire#powerrail
      Contact( #ErrorFrontal )
      S_SR(operand := #STAT_Baliza_Galibo, r1 := wire#w1)
      Coil( #Baliza )
   END_RUNG
   RUNG wire#powerrail
      Contact( #EstadoZona.Rearme_CBx )
   END_RUNG wire#w1
   RUNG wire#powerrail
      Contact( #Rearmar_ConMesaLibre )
   END_RUNG wire#w1
   // the same network as SCL:
   IF #ErrorFrontal THEN
       #STAT_Baliza_Galibo := TRUE;   // SR flip-flop
   END_IF;
   IF #EstadoZona.Rearme_CBx OR #Rearmar_ConMesaLibre THEN #STAT_Baliza_Galibo := FALSE; END_IF;
   #Baliza := #STAT_Baliza_Galibo;
END_REGION

REGION Network 28: SINOPTICO >>> Señales
   RUNG wire#powerrail
      Contact( "ON" )
      wire#w1
      Contact( #pHs_Frontal_1 )
      Coil( "DB908_Sinoptico".Galibo_Señal[#NumGalibo].Front_1 )
   END_RUNG
   RUNG wire#w1
      Contact( #pHs_Frontal_2 )
      Coil( "DB908_Sinoptico".Galibo_Señal[#NumGalibo].Front_2 )
   END_RUNG
   RUNG wire#w1
      Contact( #pHs_Frontal_3 )
      Coil( "DB908_Sinoptico".Galibo_Señal[#NumGalibo].Front_3 )
   END_RUNG
   RUNG wire#w1
      Contact( #pHs_LecturaDelantera_Des1 )
      Coil( "DB908_Sinoptico".Galibo_Señal[#NumGalibo].Frontal_Del_1 )
   END_RUNG
   RUNG wire#w1
      Contact( #pHs_LecturaDelantera_Des2 )
      Coil( "DB908_Sinoptico".Galibo_Señal[#NumGalibo].Frontal_Del_2 )
   END_RUNG
   RUNG wire#w1
      Contact( #pHs_LecturaDelantera_Error )
      Coil( "DB908_Sinoptico".Galibo_Señal[#NumGalibo].Frontal_Del_Err )
   END_RUNG
   RUNG wire#w1
      Contact( #pHs_LecturaTrasera_Des1 )
      Coil( "DB908_Sinoptico".Galibo_Señal[#NumGalibo].Frontal_Tra_1 )
   END_RUNG
   RUNG wire#w1
      Contact( #pHs_LecturaTrasera_Des2 )
      Coil( "DB908_Sinoptico".Galibo_Señal[#NumGalibo].Frontal_Tra_2 )
   END_RUNG
   RUNG wire#w1
      Contact( #pHs_LecturaTrasera_Error )
      Coil( "DB908_Sinoptico".Galibo_Señal[#NumGalibo].Frontal_Tra_Err )
   END_RUNG
   // the same network as SCL:
   "DB908_Sinoptico".Galibo_Señal[#NumGalibo].Front_1 := "ON" AND #pHs_Frontal_1;
   "DB908_Sinoptico".Galibo_Señal[#NumGalibo].Front_2 := "ON" AND #pHs_Frontal_2;
   "DB908_Sinoptico".Galibo_Señal[#NumGalibo].Front_3 := "ON" AND #pHs_Frontal_3;
   "DB908_Sinoptico".Galibo_Señal[#NumGalibo].Frontal_Del_1 := "ON" AND #pHs_LecturaDelantera_Des1;
   "DB908_Sinoptico".Galibo_Señal[#NumGalibo].Frontal_Del_2 := "ON" AND #pHs_LecturaDelantera_Des2;
   "DB908_Sinoptico".Galibo_Señal[#NumGalibo].Frontal_Del_Err := "ON" AND #pHs_LecturaDelantera_Error;
   "DB908_Sinoptico".Galibo_Señal[#NumGalibo].Frontal_Tra_1 := "ON" AND #pHs_LecturaTrasera_Des1;
   "DB908_Sinoptico".Galibo_Señal[#NumGalibo].Frontal_Tra_2 := "ON" AND #pHs_LecturaTrasera_Des2;
   "DB908_Sinoptico".Galibo_Señal[#NumGalibo].Frontal_Tra_Err := "ON" AND #pHs_LecturaTrasera_Error;
END_REGION

REGION Network 29: SINOPTICO >>> RODILLOS >>> Codigo >>> Profundidad
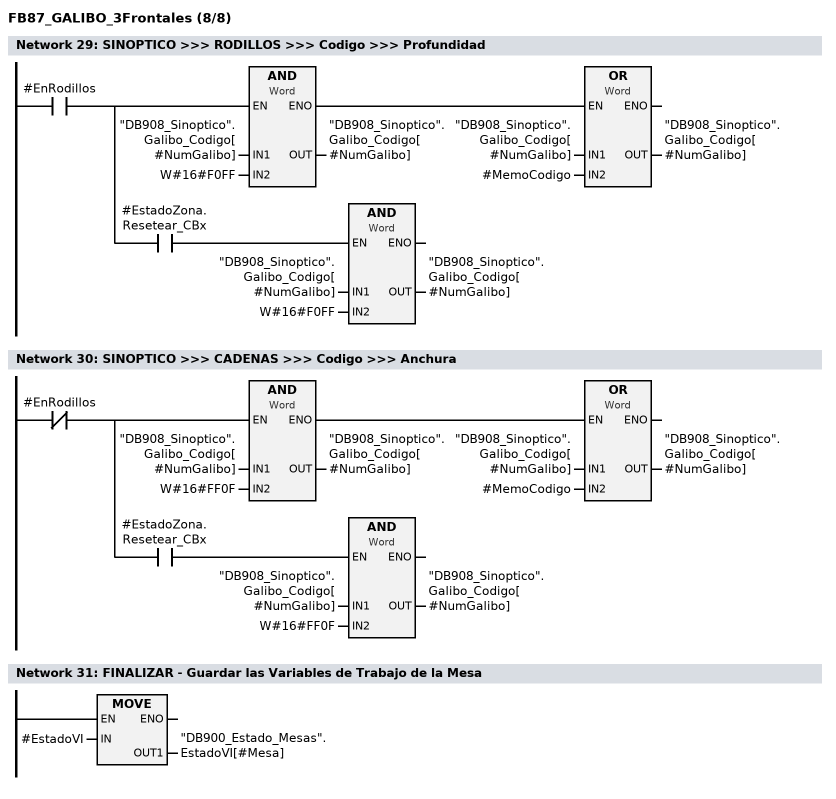
   IF #EnRodillos THEN
       "DB908_Sinoptico".Galibo_Codigo[#NumGalibo] := "DB908_Sinoptico".Galibo_Codigo[#NumGalibo] AND W#16#F0FF;
       "DB908_Sinoptico".Galibo_Codigo[#NumGalibo] := "DB908_Sinoptico".Galibo_Codigo[#NumGalibo] OR #MemoCodigo;
   END_IF;
   IF #EnRodillos AND #EstadoZona.Resetear_CBx THEN
       "DB908_Sinoptico".Galibo_Codigo[#NumGalibo] := "DB908_Sinoptico".Galibo_Codigo[#NumGalibo] AND W#16#F0FF;
   END_IF;
END_REGION

REGION Network 30: SINOPTICO >>> CADENAS >>> Codigo >>> Anchura
   IF NOT #EnRodillos THEN
       "DB908_Sinoptico".Galibo_Codigo[#NumGalibo] := "DB908_Sinoptico".Galibo_Codigo[#NumGalibo] AND W#16#FF0F;
       "DB908_Sinoptico".Galibo_Codigo[#NumGalibo] := "DB908_Sinoptico".Galibo_Codigo[#NumGalibo] OR #MemoCodigo;
   END_IF;
   IF NOT #EnRodillos AND #EstadoZona.Resetear_CBx THEN
       "DB908_Sinoptico".Galibo_Codigo[#NumGalibo] := "DB908_Sinoptico".Galibo_Codigo[#NumGalibo] AND W#16#FF0F;
   END_IF;
END_REGION

REGION Network 31: FINALIZAR - Guardar las Variables de Trabajo de la Mesa
   RUNG wire#powerrail
      Move(in := #EstadoVI, out1 => "DB900_Estado_Mesas".EstadoVI[#Mesa])
   END_RUNG
   // the same network as SCL:
   "DB900_Estado_Mesas".EstadoVI[#Mesa] := #EstadoVI;
END_REGION
END_FUNCTION_BLOCK
